PROGRAM RUN_TESTS
VAR
    CbTest    :    FB_CircuitBreaker_Test;
END_VAR

TcUnit.RUN();

END_PROGRAM

(* stored: Version 1.1.0.1, ProductVersion 3.1.4022.18
   POU RUN_TESTS: Id {e6fc24fd-e279-490c-8a71-fd69372c3aaa}, SpecialFunc None *)
